FUNCTION ARR_MIN (* Array Minimum *)
  (* Standard: 61499-1 *)
  (* Version 1.0, 2026-01-23, Franz Höpfinger, Andreas Demmler Fahrzeugbau, inspired by MIN in IEC 61131 Paper *)
  PACKAGE logiBUS::utils::dyn_arr;
  IMPORT eclipse4diac::core::TypeHash;
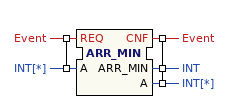
  EVENT_INPUT
    REQ WITH A;
  END_EVENT
  EVENT_OUTPUT
    CNF WITH ARR_MIN, A;
  END_EVENT
  VAR_OUTPUT
    ARR_MIN : INT;
  END_VAR
  VAR_IN_OUT
    A : ARRAY [*] OF INT; (* Input *)
  END_VAR
  BODY IN ST:
PACKAGE logiBUS::utils::dyn_arr;

(* Array Minimum *)
FUNCTION ARR_MIN : INT

VAR_IN_OUT
	A : ARRAY[*] OF INT; // Input
END_VAR

VAR_TEMP
	i : INT;
	currentMin : INT;
END_VAR

i := LOWER_BOUND(A, 1);
currentMin := A[i];
FOR i := LOWER_BOUND(A,1) + 1 TO UPPER_BOUND(A,1) DO
	currentMin := MIN(A[i], currentMin);

END_FOR;
ARR_MIN := currentMin;

END_FUNCTION
  END_BODY
END_FUNCTION
